// TIA Portal V16 export
// export: Created 2024-03-28T09:48:21.5586508Z, ExportSetting WithDefaults, DisplayName Totally Integrated Automation Portal, DisplayVersion V16, DisplayName TIA Portal Version Control Interface, DisplayVersion V16, DisplayName TIA Portal Openness, DisplayVersion V16, DisplayName STEP 7 Professional, DisplayVersion V16, DisplayName STEP 7 Safety, DisplayVersion V16, DisplayName WinCC Advanced, DisplayVersion V16
TYPE "UR__T2O_Robot"
// stored: IsFailsafeCompliant false
   STRUCT
      "Controller major version" : USInt;
      "Controller minor version" : USInt;
      Reserved { ExternalAccessible := 'False'; ExternalVisible := 'False'; ExternalWritable := 'False'} : UInt;
      "Robot mode" : USInt;
      "Real time machine seconds" : USInt;
      "Real time machine milliseconds" : UInt;
      "Real time machine minutes" : USInt;
      "Real time machine hours" : USInt;
      "Real time machine days" : UInt;
      "Robot current [A]" : Real;
      "PW: Is power on" : Bool;
      "PR: Is program running" : Bool;
      "TB: Is teach button pressed" : Bool;
      "PB: Is power button pressed" : Bool;
      Reserved_4 { ExternalAccessible := 'False'; ExternalVisible := 'False'; ExternalWritable := 'False'} : Bool;
      Reserved_5 { ExternalAccessible := 'False'; ExternalVisible := 'False'; ExternalWritable := 'False'} : Bool;
      Reserved_6 { ExternalAccessible := 'False'; ExternalVisible := 'False'; ExternalWritable := 'False'} : Bool;
      Reserved_7 { ExternalAccessible := 'False'; ExternalVisible := 'False'; ExternalWritable := 'False'} : Bool;
      Reserved_8_15 { ExternalAccessible := 'False'; ExternalVisible := 'False'; ExternalWritable := 'False'} : USInt;
      Reserved_16_31 { ExternalAccessible := 'False'; ExternalVisible := 'False'; ExternalWritable := 'False'} : UInt;
      "Speed slider fraction" : Real;
   END_STRUCT;
END_TYPE
